// TIA Portal V15.1 export
// export: Created 2024-06-21T08:40:46.8353959Z, ExportSetting WithDefaults, DisplayName Totally Integrated Automation Portal, DisplayVersion V15.1 Update 5, DisplayName TIA Portal Openness, DisplayVersion V15.1 Update 5, DisplayName SINAMICS Startdrive Advanced, DisplayVersion V15.1, DisplayName G130, G150, S120, S150, SINAMICS MV, S210, DisplayVersion V15.1, DisplayName G110M, G120, G120C, G120D, G120P, DisplayVersion V15.1, DisplayName STEP 7 Professional, DisplayVersion V15.1 Update 5, DisplayName STEP 7 Safety, DisplayVersion V15.1, DisplayName WinCC Professional, DisplayVersion V15.1 Update 5, DisplayName SIMATIC Visualization Architect, DisplayVersion V15.1
DATA_BLOCK "_209220ZS01AEAK"   // DB371
{ S7_Optimized_Access := 'FALSE' }
AUTHOR : VCC
VERSION : 0.1
// stored: AutoNumber false, DBAccessibleFromOPCUA true, IsOnlyStoredInLoadMemory false, IsWriteProtectedInAS false
   VAR RETAIN
      AB_AK01E1QM12 { ExternalAccessible := 'False'; ExternalVisible := 'False'; ExternalWritable := 'False'} : Bool;   // 400VAC - Overload protection MoviDrive chain Mode Zone 220
      AB_AK01E1QM13 { ExternalAccessible := 'False'; ExternalVisible := 'False'; ExternalWritable := 'False'} : Bool;   // 400VAC - Overload protection MoviFit chain Mode Zone 220
      AB_AK04E1QM140 { ExternalAccessible := 'False'; ExternalVisible := 'False'; ExternalWritable := 'False'} : Bool;   // 400VAC - Overload protection Brake Resistor 209220CR21
      AB_AK04E1QM143 { ExternalAccessible := 'False'; ExternalVisible := 'False'; ExternalWritable := 'False'} : Bool;   // 400VAC - Overload protection Brake Resistor 209220CR23
      AA_AE01E3FS10_CH1 { ExternalAccessible := 'False'; ExternalVisible := 'False'; ExternalWritable := 'False'} : Bool;   // 24VDC Fuse - ModeZone220 - Switch / Busnode 220AX01 & 220AS10
      AA_AE01E3FS10_CH2 { ExternalAccessible := 'False'; ExternalVisible := 'False'; ExternalWritable := 'False'} : Bool;   // 24VDC Fuse - ModeZone220 - Busnode 220AX02 & 220AS11 & 220AS20
      AC_AE01E3FS11_CH1 { ExternalAccessible := 'False'; ExternalVisible := 'False'; ExternalWritable := 'False'} : Bool;   // 24VDC Fuse - ModeZone220 - RFID Reader
      AA_AE01E3FS11_CH2 { ExternalAccessible := 'False'; ExternalVisible := 'False'; ExternalWritable := 'False'} : Bool;   // 24VDC Fuse - ModeZone220 - Eco Modules
      AD_AE01E3FS10_CH1 { ExternalAccessible := 'False'; ExternalVisible := 'False'; ExternalWritable := 'False'} : Bool;   // 24VDC Fuse - ModeZone220 - Switch / Busnode 220AX01 & 220AS10
      AD_AE01E3FS10_CH2 { ExternalAccessible := 'False'; ExternalVisible := 'False'; ExternalWritable := 'False'} : Bool;   // 24VDC Fuse - ModeZone220 - Busnode 220AX02 & 220AS11 & 220AS20
      AD_AE01E3FS11_CH1 { ExternalAccessible := 'False'; ExternalVisible := 'False'; ExternalWritable := 'False'} : Bool;   // 24VDC Fuse - ModeZone220 - RFID Reader
      AD_AE01E3FS11_CH2 { ExternalAccessible := 'False'; ExternalVisible := 'False'; ExternalWritable := 'False'} : Bool;   // 24VDC Fuse - ModeZone220 - Eco Modules
      AB_AK02E3FS56_CH1 { ExternalAccessible := 'False'; ExternalVisible := 'False'; ExternalWritable := 'False'} : Bool;   // 24VDC Fuse - General - Movidrives AK03 Mode Zone 220
      AA_AK02E3FS200_CH1 { ExternalAccessible := 'False'; ExternalVisible := 'False'; ExternalWritable := 'False'} : Bool;   // 24VDC Fuse - ModeZone 220 - DI/DO 220AX01 & 220AS10
      AA_AK02E3FS200_CH2 { ExternalAccessible := 'False'; ExternalVisible := 'False'; ExternalWritable := 'False'} : Bool;   // 24VDC Fuse - ModeZone 220 - DI/DO 220AX02 & 220AS11 & 220AS20
      AA_AK02E3FS201_CH1 { ExternalAccessible := 'False'; ExternalVisible := 'False'; ExternalWritable := 'False'} : Bool;   // 24VDC Fuse - ModeZone 220 - F-DI/F-DO 220AX01 & 220AS10
      AA_AK02E3FS201_CH2 { ExternalAccessible := 'False'; ExternalVisible := 'False'; ExternalWritable := 'False'} : Bool;   // 24VDC Fuse - ModeZone 220 - F-DI/F-DO 220AX02 & 220AS11 & 220AS20
      AB_AK02E3FS203_CH1 { ExternalAccessible := 'False'; ExternalVisible := 'False'; ExternalWritable := 'False'} : Bool;   // 24VDC Fuse - ModeZone 220 - Movifit Chain 1
      AD_AK02E3FS56_CH1 { ExternalAccessible := 'False'; ExternalVisible := 'False'; ExternalWritable := 'False'} : Bool;   // 24VDC Fuse - General - Movidrives AK03 Mode Zone 220
      AD_AK02E3FS200_CH1 { ExternalAccessible := 'False'; ExternalVisible := 'False'; ExternalWritable := 'False'} : Bool;   // 24VDC Fuse - ModeZone 220 - DI/DO 220AX01 & 220AS10
      AD_AK02E3FS200_CH2 { ExternalAccessible := 'False'; ExternalVisible := 'False'; ExternalWritable := 'False'} : Bool;   // 24VDC Fuse - ModeZone 220 - DI/DO 220AX02 & 220AS11 & 220AS20
      AD_AK02E3FS201_CH1 { ExternalAccessible := 'False'; ExternalVisible := 'False'; ExternalWritable := 'False'} : Bool;   // 24VDC Fuse - ModeZone 220 - F-DI/F-DO 220AX01 & 220AS10
      AD_AK02E3FS201_CH2 { ExternalAccessible := 'False'; ExternalVisible := 'False'; ExternalWritable := 'False'} : Bool;   // 24VDC Fuse - ModeZone 220 - F-DI/F-DO 220AX02 & 220AS11 & 220AS20
      AD_AK02E3FS203_CH1 { ExternalAccessible := 'False'; ExternalVisible := 'False'; ExternalWritable := 'False'} : Bool;   // 24VDC Fuse - ModeZone 220 - Movifit Chain 1
      AK01E1QM12AlarmABCondition { ExternalAccessible := 'False'; ExternalVisible := 'False'; ExternalWritable := 'False'} : Bool;   // Alarm AB condition
      AK01E1QM13AlarmABCondition { ExternalAccessible := 'False'; ExternalVisible := 'False'; ExternalWritable := 'False'} : Bool;   // Alarm AB condition
      AK04E1QM140AlarmABCondition { ExternalAccessible := 'False'; ExternalVisible := 'False'; ExternalWritable := 'False'} : Bool;   // Alarm AB condition
      AK04E1QM143AlarmABCondition { ExternalAccessible := 'False'; ExternalVisible := 'False'; ExternalWritable := 'False'} : Bool;   // Alarm AB condition
      AE01E3FS10_CH1AlarmABCondition { ExternalAccessible := 'False'; ExternalVisible := 'False'; ExternalWritable := 'False'} : Bool;   // Alarm AB condition
      AE01E3FS10_CH2AlarmABCondition { ExternalAccessible := 'False'; ExternalVisible := 'False'; ExternalWritable := 'False'} : Bool;   // Alarm AB condition
      AE01E3FS11_CH2AlarmABCondition { ExternalAccessible := 'False'; ExternalVisible := 'False'; ExternalWritable := 'False'} : Bool;   // Alarm AB condition
      AK02E3FS56_CH1AlarmABCondition { ExternalAccessible := 'False'; ExternalVisible := 'False'; ExternalWritable := 'False'} : Bool;   // Alarm AB condition
      AK02E3FS200_CH1AlarmABCondition { ExternalAccessible := 'False'; ExternalVisible := 'False'; ExternalWritable := 'False'} : Bool;   // Alarm AB condition
      AK02E3FS200_CH2AlarmABCondition { ExternalAccessible := 'False'; ExternalVisible := 'False'; ExternalWritable := 'False'} : Bool;   // Alarm AB condition
      AK02E3FS201_CH1AlarmABCondition { ExternalAccessible := 'False'; ExternalVisible := 'False'; ExternalWritable := 'False'} : Bool;   // Alarm AB condition
      AK02E3FS201_CH2AlarmABCondition { ExternalAccessible := 'False'; ExternalVisible := 'False'; ExternalWritable := 'False'} : Bool;   // Alarm AB condition
      AK02E3FS203_CH1AlarmABCondition { ExternalAccessible := 'False'; ExternalVisible := 'False'; ExternalWritable := 'False'} : Bool;   // Alarm AB condition
      H_209000AK01E1QM12IAnim : Word;   // HMI Animation of the icon
      H_209000AK01E1QM13IAnim : Word;   // HMI Animation of the icon
      H_209000AK04E1QM140IAnim : Word;   // HMI Animation of the icon
      H_209000AK04E1QM143IAnim : Word;   // HMI Animation of the icon
      H_209000AE01E3FS10_CH1IAnim : Word;   // HMI Animation of the icon
      H_209000AE01E3FS10_CH2IAnim : Word;   // HMI Animation of the icon
      H_209000AE01E3FS11_CH1IAnim : Word;   // HMI Animation of the icon
      H_209000AE01E3FS11_CH2IAnim : Word;   // HMI Animation of the icon
      H_209000AK02E3FS56_CH1IAnim : Word;   // HMI Animation of the icon
      H_209000AK02E3FS200_CH1IAnim : Word;   // HMI Animation of the icon
      H_209000AK02E3FS200_CH2IAnim : Word;   // HMI Animation of the icon
      H_209000AK02E3FS201_CH1IAnim : Word;   // HMI Animation of the icon
      H_209000AK02E3FS201_CH2IAnim : Word;   // HMI Animation of the icon
      H_209000AK02E3FS202_CH1IAnim : Word;   // HMI Animation of the icon
      H_209000AK02E3FS202_CH2IAnim : Word;   // HMI Animation of the icon
      H_209000AK02E3FS203_CH1IAnim : Word;   // HMI Animation of the icon
      H_209000AK02E3FS203_CH2IAnim : Word;   // HMI Animation of the icon
      H_DBnr : Int;   // DB number
      H_Anim : Word;   // Animation
      AlarmA { ExternalAccessible := 'False'; ExternalVisible := 'False'; ExternalWritable := 'False'} : Bool;   // Alarm A
      AlarmB { ExternalAccessible := 'False'; ExternalVisible := 'False'; ExternalWritable := 'False'} : Bool;   // Alarm B
      AlarmC { ExternalAccessible := 'False'; ExternalVisible := 'False'; ExternalWritable := 'False'} : Bool;   // Alarm C
      AlarmD { ExternalAccessible := 'False'; ExternalVisible := 'False'; ExternalWritable := 'False'} : Bool;   // Alarm D
      AlarmABCondition { ExternalAccessible := 'False'; ExternalVisible := 'False'; ExternalWritable := 'False'} : Bool;   // Alarm AB condition
   END_VAR
BEGIN
END_DATA_BLOCK
